# EPICS substitutions: iocBoot/iocTomoScan_2BMB/tomoScanStep.substitutions
file "$(TOP)/db/tomoScan_step.template"
{
pattern
{  P,       R}
{2bmb:, TomoScan:}
}
